# B&R Automation Studio project lab-2.1
Automation Studio 

## Configuration SampleText

### IoMap.iom - 4PP065_0571_P74/IoMap.iom
```iecst
VAR_CONFIG
	Cyclic#1.gAxis01_DrvIf.iLifeCnt AT %IB."8I64xxxxxxx.00x-1".SDC_LifeCnt;
	Cyclic#1.gAxis01_DrvIf.iDrvOK AT %IX."8I64xxxxxxx.00x-1".ETAD_Input_Bool_02;
	Cyclic#1.gAxis01_DrvIf.oSetTime AT %QW."8I64xxxxxxx.00x-1".SDC_SetTime;
	Cyclic#1.gAxis01_DiDoIf.iLifeCntDriveReady AT %IB."8I64xxxxxxx.00x-1".SDC_LifeCnt;
	Cyclic#1.gAxis01_DiDoIf.iLifeCntDriveEnable AT %IB."8I64xxxxxxx.00x-1".SDC_LifeCnt;
	Cyclic#1.gAxis01_DiDoIf.oDriveEnable AT %QX."8I64xxxxxxx.00x-1".CMDD_Output_Bool_00;
	Cyclic#1.gAxis01_ModuleOk AT %QX."8I64xxxxxxx.00x-1".CMDD_Output_Bool_01;
	Cyclic#1.gAxis01_ModuleOk AT %QX."8I64xxxxxxx.00x-1".CMDD_Output_Bool_02;
	Cyclic#1.gAxis01_ModuleOk AT %IX."8I64xxxxxxx.00x-1".ModuleOk;
	Cyclic#1.gAxis01_DiDoIf.oDriveEnable AT %QX."8I64xxxxxxx.00x-1".CMDD_Output_Bool_03;
	Cyclic#1.gAxis01_DiDoIf.iDriveReady AT %IX."8I64xxxxxxx.00x-1".ETAD_Input_Bool_02;
	::Program:driveSMFB.state AT %IW."8I64xxxxxxx.00x-1".ETAD_Input;
	::Program:driveSMFB.command AT %QW."8I64xxxxxxx.00x-1".CMDD_Output;
	::Program:doorSMFB.direction AT %IX."X20DI9371".DigitalInput01;
	::Program:doorSMFB.sw0 AT %IX."X20DI9371".DigitalInput02;
	::Program:doorSMFB.sw1 AT %IX."X20DI9371".DigitalInput03;
	::Program:doorSMFB.sw2 AT %IX."X20DI9371".DigitalInput04;
	::Program:doorSMFB.sw3 AT %IX."X20DI9371".DigitalInput05;
	::Program:ledSMFB.led1 AT %QX."X20DO9322".DigitalOutput02;
	::Program:ledSMFB.led2 AT %QX."X20DO9322".DigitalOutput03;
	::Program:ledSMFB.led3 AT %QX."X20DO9322".DigitalOutput04;
	::Program:ledSMFB.led4 AT %QX."X20DO9322".DigitalOutput05;
	Cyclic#1.::Program:driveSMFB.speed AT %QW."8I64xxxxxxx.00x-1".LFRD_Output;
END_VAR
```

## Logical view

- Library Logical/Libraries/DriveLib (ANSIC) (no source held here)

### Program Logical/Program

#### Variables.var
```iecst
VAR
	driveSMFB : FB_DriveStateMachine := (0);
	doorSMFB : FB_DoorStateMachine := (0);
	ledSMFB : FB_LedStateMachine := (0);
END_VAR
```

#### Cyclic.c
```c
#include <bur/plctypes.h>

#ifdef _DEFAULT_INCLUDES
	#include <AsDefault.h>
#endif

void _CYCLIC ProgramCyclic(void)
{
	FB_DoorStateMachine(&doorSMFB);
	driveSMFB.speed = doorSMFB.speed;
	FB_DriveStateMachine(&driveSMFB);
	ledSMFB.state = doorSMFB.state;
	FB_LedStateMachine(&ledSMFB);
}
```

#### Init.c
```c
#include <bur/plctypes.h>

#ifdef _DEFAULT_INCLUDES
	#include <AsDefault.h>
#endif

void _INIT ProgramInit(void)
{
	driveSMFB.enable=1;
}
```

Listed in the project but not available here: Logical/Libraries/DriveLib/Types.typ, Logical/Libraries/DriveLib/Constants.var, Logical/Libraries/DriveLib/DriveLib.fun, Logical/Libraries/DriveLib/FB_DriveStateMachine.c, Logical/Libraries/DriveLib/FB_DoorStateMachine.c, Logical/Libraries/DriveLib/FB_LedStateMachine.c
